FUNCTION Convert_UINT_TO_LINT : Hresult
VAR_INPUT
	in : UINT;
	out : REFERENCE TO LINT;
END_VAR
VAR
	converted : LINT;
END_VAR

converted := UINT_TO_LINT(in);

IF (LINT_TO_UINT(converted) <> in) THEN
	Convert_UINT_TO_LINT := INCOMPATIBLE;
	RETURN;
END_IF

out := converted;

END_FUNCTION

(* stored: Version 1.1.0.1, ProductVersion 3.1.4024.12
   POU Convert_UINT_TO_LINT: Id {e34aff37-620a-410e-b095-139550b59eca}, SpecialFunc None *)
